Fanuc KAREL source: LN.kl

PROGRAM T
%NOLOCKGROUP
VAR
 v0 : REAL
 res : REAL
BEGIN
 res = LN(v0)
END T
